// Mitsubishi GX Works2 project: BIN Instruction   PLC: Q03UDV

PROGRAM MAIN
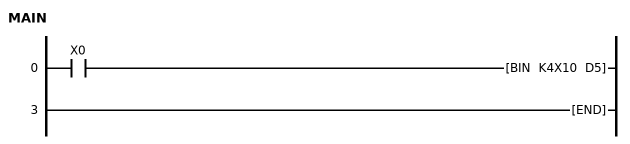
0     LD      X0
      BIN     K4X10 D5
3     END
END_PROGRAM
